# B&R Automation Studio project Parker_BMM_ST_V5_3147_V12 (part 4)

```iecst
(*Temperature fix and parameter type *)

TYPE
	Zones_Status_typ : 	STRUCT
		idxNotNormal : USINT;
		bNotNormal : BOOL;
		bAlarmHeatNormal : ARRAY[0..MAX_IDX_ZONE]OF BOOL;
		idxBroken : USINT;
		bBroken : BOOL; (*machine sensor broken*)
		SensorBroken : ARRAY[0..MAX_IDX_ZONE]OF BOOL; (*zone sensor broken*)
		bLowInternal : BOOL;
		idxLow : USINT;
		bLow : BOOL; (*machine alarm low*)
		AlmLow : ARRAY[0..MAX_IDX_ZONE]OF BOOL; (*zone alarm low*)
		idxHigh : USINT;
		bHigh : BOOL; (*machine alarm high*)
		AlmHigh : ARRAY[0..MAX_IDX_ZONE]OF BOOL; (*zone alarm high*)
		idxSwitchoff : USINT;
		bSwitchOff : BOOL; (*machine temperature high -switch off*)
		TempSwitchOff : ARRAY[0..MAX_IDX_ZONE]OF BOOL; (*temperature too high -- switch off*)
		idxFreeze : USINT;
		bFreeze : BOOL; (*machine heating exception*)
		TempFreeze : ARRAY[0..MAX_IDX_ZONE]OF BOOL; (*heating exception -- temperature freeze*)
		Tuning : ARRAY[0..MAX_IDX_ZONE]OF BOOL; (*zone is tuning*)
		TuneOk : ARRAY[0..MAX_IDX_ZONE]OF BOOL; (*zone tuning ok*)
		TuneStatus : ARRAY[0..MAX_IDX_ZONE]OF UINT; (*zone tune step and error feedback*)
		PreHeatingOk : ARRAY[0..MAX_IDX_ZONE]OF BOOL; (*zone pre-heating ok or not*)
		okToHeat : ARRAY[0..MAX_IDX_ZONE]OF BOOL; (*function need*)
		okToFree : ARRAY[0..MAX_IDX_ZONE]OF BOOL; (*function need*)
		okToFreeEnd : ARRAY[0..MAX_IDX_ZONE]OF BOOL; (*function need*)
		okToCool : ARRAY[0..MAX_IDX_ZONE]OF BOOL; (*function need*)
		okToCoolEnd : ARRAY[0..MAX_IDX_ZONE]OF BOOL; (*function need*)
		Out : ARRAY[0..MAX_IDX_ZONE]OF INT;
	END_STRUCT;
END_TYPE
```

### Global.var - Global variable
```iecst
(*global variables*)
VAR
	gAccuLinear : DCDT_typ;
	gAlarm : Alarm_typ;
	gAxisCtrl : ARRAY[0..MAX_AXIS_NUM] OF Axis_Ctrl_typ;
	gControlInfo : Control_Info_typ;
	gDS1119_Axis : ARRAY[0..MAX_AXIS_NUM] OF DS;
END_VAR
VAR RETAIN
	gExtruderA : Extruder_Ctrl_typ;
	gExtruderB : Extruder_Ctrl_typ;
	gExtruderC : Extruder_Ctrl_typ;
	gExtruderD : Extruder_Ctrl_typ := (0);
	gExtruderVisu : Extruder_Ctrl_typ;
	gH_IO : H_Zone_typ := (0);
END_VAR
VAR
	gHardWare : HardWare_typ;
END_VAR
VAR RETAIN
	gHeatingPlan : Heating_Plan_typ := (0);
END_VAR
VAR
	gImply : Imply_typ;
	gMachineFix : Machine_Fix_typ;
	gMachineIn : Machine_In_typ;
	gMachineInfo : Machine_Info_typ;
	gMachineOut : Machine_Out_typ;
	gMachinePara : Machine_Para_typ;
END_VAR
VAR RETAIN
	gMachineWorkDays : UDINT;
	gMachineStopDays : UDINT;
	gMachineWorkTime : UDINT;
	gMacOption : Machine_Option_typ;
	gBatchInfo : Batch_Info_typ;
END_VAR
VAR
	gMacTimer : Machine_Timer_typ;
	gPanelObj : Panel_Basic_typ;
	gPROCESS_info : Process_Status_typ;
	gPwd : Pwd_typ;
	gRecipeOperate : Recipe_Operate_typ;
	gScreenShot : ScreenShotObj_typ;
	gServoLinear : DCDT_typ;
END_VAR
VAR RETAIN
	gSPC_Current : SPC_Unit_typ;
	gT_Par : Temp_Ctrl_typ := (0);
END_VAR
VAR
	gThickData : Thick_Data_typ;
	gTempData : ARRAY[0..100] OF DINT;
	gThickFix : Thick_Fix_typ;
	gThickIO : Thick_IO_typ;
END_VAR
VAR RETAIN
	gThickProf : Profile_typ;
END_VAR
VAR
	gTKauto : task_status_type;
	gTKcalib : task_status_type;
	gTKmanual : task_status_type;
	gUSB_1 : USB_Device_typ;
	gUSB_2 : USB_Device_typ;
	gUserFix : User_Fix_typ;
	gUserFix_new : User_Fix_new_typ;
	gUserPara : User_Para_typ;
END_VAR
VAR RETAIN
	gCycleTimes : UDINT;
	gCycleTimesL : UDINT;
	gCycleTimesR : UDINT;
END_VAR
VAR CONSTANT
	LED_OFF : USINT := 0;
	LED_ON : USINT := 1;
	LED_QUICK_BLINK : USINT := 3;
	LED_SLOW_BLINK : USINT := 2;
END_VAR
VAR
	LMold : Mold_typ;
	RMold : Mold_typ;
END_VAR
(*Test Pump*)
VAR
	btnTesetPQ1 : BOOL;
	btnTesetPQ : BOOL;
END_VAR
(*Servo Axis*)
VAR
	gAxisClampL : ACP10AXIS_typ;
	gAxisClampR : ACP10AXIS_typ;
	gAxisCarriageL : ACP10AXIS_typ;
	gAxisCarriageR : ACP10AXIS_typ;
	gAxisBlowPinL : ACP10AXIS_typ;
	gAxisBlowPinR : ACP10AXIS_typ;
	gAxisBlowPin2L : ACP10AXIS_typ;
	gAxisBlowPin2R : ACP10AXIS_typ;
	gAxisTransferL : ACP10AXIS_typ;
	gAxisTransferR : ACP10AXIS_typ;
	gAxisUpDnL : ACP10AXIS_typ;
	gAxisUpDnR : ACP10AXIS_typ;
	gAxisExtrlift : ACP10AXIS_typ;
	gAxisThick : ACP10AXIS_typ;
END_VAR
(*Extruder Inverter Powerlink*)
VAR
	ExtruderA_Retain : {REDUND_UNREPLICABLE} Extruder_Basic_typ := (0); (*wzq*)
	ExtruderB_Retain : {REDUND_UNREPLICABLE} Extruder_Basic_typ := (0); (*wzq*)
	ExtruderC_Retain : Extruder_Basic_typ;
	ExtruderV_Retain : Extruder_Basic_typ;
	gExtruderACtrl : Inverter_Ctrl_typ;
	gExtruderBCtrl : Inverter_Ctrl_typ;
	gExtruderCCtrl : Inverter_Ctrl_typ;
	gExtruderVCtrl : Inverter_Ctrl_typ;
END_VAR
(*Robot Time*)
VAR
	LRobotCarriageTime : TOF_10ms;
	RobotCarriageTime : TOF_10ms;
	LRobotClampTime : TOF_10ms;
	RobotClampTime : TOF_10ms;
END_VAR
(*Insert your comment here.*)
VAR
	LRobotClampTimePara : UDINT;
	RobotClampTimePara : UDINT;
	LRobotCarriageTimePara : UDINT;
	RobotCarriageTimePara : UDINT;
	usScaleIndex : USINT;
	gLClampOpnFlag_Calib : USINT;
	gRClampOpnFlag_Calib : USINT;
	ParisonSacleDown : DINT;
	ParisonSacleUp : DINT;
	ParisonSacleDown_Old : DINT;
	ParisonSacleUp_Old : DINT;
	ParisonSacleDownFlag : BOOL;
	ParisonSacleUpFlag : BOOL;
	ParisonSacleDownFlag_Old : BOOL;
	ParisonSacleUpFlag_Old : BOOL;
	gLevelTooLow : BOOL;
	gExtruderTempLow_HMIFlag : BOOL;
	gTempfirstHeatOK : DINT;
	gTempfirstHeatOK_Flag : BOOL;
	gPasswordLogout : BOOL;
	gAcs380Ctrl : Acs380Ctl_type;
	gEnableAll_HMI : BOOL;
	gDisableAll_HMI : BOOL;
	gExtruderHMI_Enable : ARRAY[0..NUM_ACS380_MINUS_ONE] OF BOOL;
END_VAR
VAR CONSTANT
	NUM_ACS380_MINUS_ONE : USINT := 4; (*Acs380数量-1*)
END_VAR
VAR
	ExIndex : USINT;
	gExSPC : ARRAY[0..19] OF ExSPC_typ;
	gExSPC_Clear : BOOL;
	gAxisPwr : ACP10AXIS_typ;
	gMotorTrace : MotorTrace_typ;
	gAxisCarriageR_1 : ACP10AXIS_typ;
END_VAR
```

### Library Logical/Libraries/SimpFun (IEC, version 2.10.0) - Get time function library
Depends on: AsIO, AsString, AsTime, runtime

#### DateTimeString.st
```iecst
FUNCTION_BLOCK DateTimeString
(* Implementation of ST_DateTimeString *)

(*
//******************************************************************************************************//
//		 B & R - Bernecker and Rainer China 		              										              //
//******************************************************************************************************//
// Library Name:	SimpFun																			                       //
// Function Name:	DateTimeString																		                    //
// Autor:			B&R 						      	  										                          //
//------------------------------------------------------------------------------------------------------//
// Description: 	Print Different type Date and Time									  				              //
//-------------------------------------------------------------------------------------------------------//

//-------------------------------------------------------------------------------------------------------//
//	History:	6.Nov.2008	 V1.00														                                 //
//				V1.00: Just 24 hour time mode															                     //
//*******************************************************************************************************//

//*******************************************************************************************************//
//	<|> Variable to control this task:																	                  //
//		Name							Typ					Description									                     //
//		strYYYY							STRING[4]			Save Year as STRING	type			                     //
//		strMonthM						STRING[2]			Save Month as STRING type			                     //
//		strDD							STRING[2]			Save Day as STRING type						                  //
//		strHH							STRING[2]			Save Hour as STRING type					                  //
//		strMinuteM						STRING[2]			Save Minute as STRING type				                  //
//		strSS							STRING[2]			Save Second as STRING type					                  //
//		flagAMPM						BOOL				current time is AM or PM:0=AM,1=PM			                  //
//*******************************************************************************************************//

//*******************************************************************************************************//
//  Others:																								                        //
//		V1.00:																							                        //
//			Date_Mode																					                        //
//				1:		USA date format -- DateMM-DD-YYYY_TimeHH-MM-SS								                  //
//				2:		Asia DATE format -- DateYYYY-MM-DD_TimeHH-MM-SS								                  //
//				others:	Default format -- DateDD-MM-YYYY_TimeHH-MM-SS							                  //
//*******************************************************************************************************//
*)

IF (enable = 1) THEN

	DTGetTime_0.enable := 1;
	DTGetTime_0();

	DT_TO_DTStructure(DTGetTime_0.DT1, ADR(currentTime));

	strcpy(ADR(DisplayString),ADR('Date'));								(* DisplayString = "Date" *)

	itoa(currentTime.year, ADR(strYYYY));								(* string -- "YYYY" *)
	itoa(currentTime.month, ADR(strMonthM));							(* string -- "MM: month" *)
	itoa(currentTime.day, ADR(strDD));									(* string -- "DD" *)

	CASE Date_Mode OF
		1:		(* USA date format -- MM-DD-YYYY *)

			(***** ADD MM   Month *****)
			IF currentTime.month <= 9 THEN
				strcat(ADR(DisplayString), ADR('0'));					(* DisplayString = "Date0" *)
			END_IF
			strcat(ADR(DisplayString), ADR(strMonthM));					(* DisplayString = "DateMM" *)
			strcat(ADR(DisplayString), ADR('-'));						(* DisplayString = "DateMM-" *)

			(***** ADD DD *****)
			IF currentTime.day <= 9 THEN
				strcat(ADR(DisplayString), ADR('0'));					(* DisplayString = "DateMM-0" *)
			END_IF
			strcat(ADR(DisplayString), ADR(strDD));						(* DisplayString = "DateMM-DD" *)
			strcat(ADR(DisplayString), ADR('-'));						(* DisplayString = "DateMM-DD-" *)

			(***** ADD YYYY *****)
			strcat(ADR(DisplayString), ADR(strYYYY));					(* DisplayString = "DateMM-DD-YYYY" *)

		2:		(* Asia date format -- YYYY-MM-DD *)

			(***** ADD YYYY *****)
			strcat(ADR(DisplayString), ADR(strYYYY));					(* DisplayString = "DateYYYY" *)
			strcat(ADR(DisplayString), ADR('-'));						(* DisplayString = "DateYYYY-" *)

			(***** ADD MM   Month *****)
			IF currentTime.month <= 9 THEN
				strcat(ADR(DisplayString), ADR('0'));					(* DisplayString = "DateYYYY-0" *)
			END_IF
			strcat(ADR(DisplayString), ADR(strMonthM));					(* DisplayString = "DateYYYY-MM" *)
			strcat(ADR(DisplayString), ADR('-'));						(* DisplayString = "DateYYYY-MM-" *)

			(***** ADD DD *****)
			IF currentTime.day <= 9 THEN
				strcat(ADR(DisplayString), ADR('0'));					(* DisplayString = "DateYYYY-MM-0" *)
			END_IF
			strcat(ADR(DisplayString), ADR(strDD));						(* DisplayString = "DateYYYY-MM-DD" *)

		ELSE	(* Default format -- DD-MM-YYYY *)

			(***** ADD DD *****)
			IF currentTime.day <= 9 THEN
				strcat(ADR(DisplayString), ADR('0'));					(* DisplayString = "Date0" *)
			END_IF
			strcat(ADR(DisplayString), ADR(strDD));						(* DisplayString = "DateDD" *)
			strcat(ADR(DisplayString), ADR('-'));						(* DisplayString = "DateDD-" *)

			(***** ADD MM   Month *****)
			IF currentTime.month <= 9 THEN
				strcat(ADR(DisplayString), ADR('0'));					(* DisplayString = "DateDD-0" *)
			END_IF
			strcat(ADR(DisplayString), ADR(strMonthM));					(* DisplayString = "DateDD-MM" *)
			strcat(ADR(DisplayString), ADR('-'));						(* DisplayString = "DateDD-MM-" *)

			(***** ADD YYYY *****)
			strcat(ADR(DisplayString), ADR(strYYYY));					(* DisplayString = "DateDD-MM-YYYY" *)

	END_CASE

	strcat(ADR(DisplayString),ADR('_Time'));							(* DisplayString = "DateDD-MM-YYYY_Time" *)

	itoa(currentTime.minute, ADR(strMinuteM));							(* string -- "MM: minute" *)
	itoa(currentTime.second, ADR(strSS));								(* string -- "SS" *)

	(***** ADD HH : 24 Hour mode*****)
		IF currentTime.hour <= 9 THEN
			strcat(ADR(DisplayString), ADR('0'));						(* DisplayString = "DateDD-MM-YYYY_Time0" *)
		END_IF
		itoa(currentTime.hour, ADR(strHH));								(* string -- "HH" *)
		strcat(ADR(DisplayString), ADR(strHH));							(* DisplayString = "DateDD-MM-YYYY_TimeHH" *)
	END_IF
	strcat(ADR(DisplayString), ADR('-'));								(* DisplayString = "DateDD-MM-YYYY_TimeHH-" *)

	(***** ADD MM   minute *****)
	IF currentTime.minute <= 9 THEN
		strcat(ADR(DisplayString), ADR('0'));							(* DisplayString = "DateDD-MM-YYYY_TimeHH-0" *)
	END_IF
	strcat(ADR(DisplayString), ADR(strMinuteM));						(* DisplayString = "DateDD-MM-YYYY_TimeHH-MM" *)
	strcat(ADR(DisplayString), ADR('-'));								(* DisplayString = "DateDD-MM-YYYY_TimeHH-MM-" *)

	(***** ADD SS *****)
	IF currentTime.second <= 9 THEN
		strcat(ADR(DisplayString), ADR('0'));							(* DisplayString = "DateDD-MM-YYYY_TimeHH-MM-0" *)
	END_IF
	strcat(ADR(DisplayString), ADR(strSS));								(* DisplayString = "DateDD-MM-YYYY_TimeHH-MM-SS" *)

	StringLength := strlen(ADR(DisplayString));							(* Output StringLength -- length of the DisplayString *)

END_FUNCTION_BLOCK
```

#### IOForcingOperate.st
```iecst
FUNCTION_BLOCK IOForcingOperate
(* Implementation of IOForcingOperate *)

(*
//******************************************************************************************************//
//		 B & R - Bernecker and Rainer China 		              										              //
//******************************************************************************************************//
// Library Name:	SimpFun																			                       //
// Function Name:	IOForcingOperate																	                    //
// Autor:			B&R 						      	  										                          //
//------------------------------------------------------------------------------------------------------//
// Description: 	operate IO: Enable/disable 		 									  				              //
//------------------------------------------------------------------------------------------------------//

//------------------------------------------------------------------------------------------------------//
//	History:	 	23.Nov.2008	 V1.00														                             //

//******************************************************************************************************//

//******************************************************************************************************//
//	<|> Variable to control this task:																	                 //
//		Name						Typ						Description									                    //
//		AsIOSetForceValue_0			| AsIOSetForceValue 	| Set force value							              //
//		AsIOEnableForcing_0			| AsIOEnableForcing 	| Enable force value						              //
//		AsIODisableForcing_0		| AsIODisableForcing 	| Disable forceing							           //

//******************************************************************************************************//

//******************************************************************************************************//
//  Others:																								                       //
//		V1.00:																							                       //
			be careful: make sure EnableForcing and DisableForcing, only one is true.
//		Name						Typ						Description									                    //
		IN:
//			enable					| BOOL					| enable this function						              //
//			EnableForcing			| BOOL					| =1:this function use to enable forcing	           //
//			Value					| UDINT					| the forcing value							                 //
//			DisableForcing			| BOOL					| =1:this function use to disable forcing	           //
		OUT:
//			status					| UINT					| =0: no error								                 //
//			InForcing				| USINT					| =0: No forcing							                 //
//															  =1: Forcing to zero						                    //
//															  =2: Forcing to one						                       //

//******************************************************************************************************//
*)

IF (enable = 1) THEN
	CASE (step) OF
		0:			(* init step *)
			status := 65535;
			IF (EnableForcing = 1) THEN								(* Enable Forcing *)
				step := 10;
			ELSIF (DisableForcing = 1) THEN
				step := 30;											(* Disable Forcing *)
			END_IF

		10:			(* set force value *)
			AsIOSetForceValue_0.enable     := 1;
			AsIOSetForceValue_0.pDatapoint := ADR(DataPoint);		(* Pointer to the I/O data point name *)
			AsIOSetForceValue_0.value      := Value;

			AsIOSetForceValue_0();

			IF (AsIOSetForceValue_0.status <> 65535) THEN
				IF (AsIOSetForceValue_0.status = 0) THEN
					step := 20;
				ELSE
					status := AsIOSetForceValue_0.status;
					step := 200;									(* Error *)
				END_IF
			END_IF

		20:			(* Enable forcing *)
			AsIOEnableForcing_0.enable := 1;
			AsIOEnableForcing_0.pDatapoint := ADR(DataPoint);

			AsIOEnableForcing_0();

			IF (AsIOEnableForcing_0.status <> 65535) THEN
				IF (AsIOEnableForcing_0.status = 0) THEN
					IF (Value = 0) THEN
						InForcing := 1;
					ELSE
						InForcing := 2;
					END_IF
					step := 100;									(* Enable forcing ok *)

				ELSE
					status := AsIOEnableForcing_0.status;
					step := 200;									(* Error *)

				END_IF
			END_IF

		30:			(* Disable forcing *)
			AsIODisableForcing_0.enable := 1;
			AsIODisableForcing_0.pDatapoint := ADR(DataPoint);

			AsIODisableForcing_0();

			IF (AsIODisableForcing_0.status <> 65535) THEN
				IF (AsIODisableForcing_0.status = 0) THEN
					InForcing := 0;
					step := 100;									(* Disable forcing ok *)
				ELSE
					status := AsIODisableForcing_0.status;
					step := 200;									(* Error *)
				END_IF
			END_IF

		100:		(* Operator OK *)
			status := 0;
			step := 0;

		200: 		(* Error step *)
			(* the error number has record in status *)
			step := 0;

	END_CASE
END_IF
END_FUNCTION_BLOCK
```

#### Scaler_ActZone.st
```iecst
FUNCTION_BLOCK Scaler_ActZone
(* Implementation of Scaler_ActZone *)

IF Enable = 1 THEN
	IF (MaxInV <= MinInV) OR (MaxOutV <= MinOutV) OR (ActZoneMaxV <= ActZoneMinV) THEN

		status := 1;							(* Parameter Error: MaxInV/MaxOutV/ActZoneMaxV must larger than MinInV/MinOutV/ActZoneMinV *)
	ELSIF (ActZoneMinV < MinInV) OR (MaxInV < ActZoneMaxV) THEN
		status := 2;							(* Parameter Error: [ActZoneMinV, ActZoneMaxV] must be loacaled in [MinInV, MaxInV] *)
	ELSIF (Mode_Current = 0) AND ((MinOutV < -10) OR (MaxOutV > 10)) THEN
		status := 3;							(* Parameter Error: For Voltage Output, MaxInV and MinInV must be localed in [-10, 10] *)
	ELSIF (Mode_Current = 1) AND ((MinOutV < -20) OR (MaxOutV > 20)) THEN
		status := 4;							(* Parameter Error: For Current Output, MaxInV and MinInV must be localed in [-20, 20] *)
	ELSE										(* Parameter Correct *)
		status := 0;

		IF (SV < ActZoneMinV) THEN
			IF (Mode_Current = 0) THEN
				Out := REAL_TO_INT(INT_TO_REAL(MinOutV)*32767/10);
			ELSE
				Out := REAL_TO_INT(INT_TO_REAL(MinOutV)*32767/20);
			END_IF
		ELSIF (SV > ActZoneMaxV) THEN
			IF (Mode_Current = 0) THEN
				Out := REAL_TO_INT(INT_TO_REAL(MinOutV)*32767/10);
			ELSE
				Out := REAL_TO_INT(INT_TO_REAL(MinOutV)*32767/20);
			END_IF
		ELSE
			IF (Mode_Current = 0) THEN
				Out := REAL_TO_INT(((INT_TO_REAL(MaxOutV) - MinOutV)*(SV - MinInV)/(MaxInV - MinInV) + MinOutV)*32767/10);
			ELSE
				Out := REAL_TO_INT(((INT_TO_REAL(MaxOutV) - MinOutV)*(SV - MinInV)/(MaxInV - MinInV) + MinOutV)*32767/20);
			END_IF
		END_IF
	END_IF
END_IF
END_FUNCTION_BLOCK
```

#### SimpFun.fun
```iecst
FUNCTION_BLOCK DateTimeString
VAR
		DTGetTime_0	:DTGetTime;
		currentTime	:DTStructure;
		strYYYY	:STRING[4];
		strDD	:STRING[2];
		strHH	:STRING[2];
		strSS	:STRING[2];
		strMonthM	:STRING[2];
		strMinuteM	:STRING[2];
	END_VAR
	VAR_INPUT
		enable	:BOOL;
		Date_Mode	:USINT;
	END_VAR
	VAR_OUTPUT
		DisplayString	:STRING[80];
		StringLength	:UINT;
	END_VAR
END_FUNCTION_BLOCK
FUNCTION_BLOCK IOForcingOperate
VAR
		step	:USINT;
		AsIOSetForceValue_0	:AsIOSetForceValue;
		AsIOEnableForcing_0	:AsIOEnableForcing;
		AsIODisableForcing_0	:AsIODisableForcing;
	END_VAR
	VAR_INPUT
		enable	:BOOL;
		DataPoint	:STRING[80];
		EnableForcing	:BOOL;
		Value	:UDINT;
		DisableForcing	:BOOL;
	END_VAR
	VAR_OUTPUT
		status	:UINT;
		InForcing	:USINT;
	END_VAR
END_FUNCTION_BLOCK
FUNCTION_BLOCK Scaler_ActZone
VAR_INPUT
		Enable	:BOOL;
		MaxInV	:INT;
		MinInV	:INT;
		ActZoneMaxV	:INT;
		ActZoneMinV	:INT;
		MaxOutV	:INT;
		MinOutV	:INT;
		SV	:INT;
		Mode_Current	:BOOL;
	END_VAR
	VAR_OUTPUT
		Out	:INT;
		status	:UINT;
	END_VAR
END_FUNCTION_BLOCK
```

### Program Logical/In_Out/tk1_in (ANSIC) - task 1 fast input

#### tk1_in.c
```c
/********************************************************************
 * COPYRIGHT --  B&R China
 ********************************************************************
 * Program: tk1_in
 * File: tk1_in.c
 * Author: lijianjun
 * Created: March 06, 2013
 ********************************************************************
 * Implementation of program tk1_in --- task 1# input
 ********************************************************************/

#include <bur/plctypes.h>
#include <string.h>

#ifdef _DEFAULT_INCLUDES
#include <AsDefault.h>
#endif

#include "edge.h"               /*edge function                         */

/*************************************************************************************
     	        		I N I T U P  O F   T H E   T A S K
*************************************************************************************/
_INIT void init ( void )
{
	RTInfo_Task.enable = 1;
	RTInfo(&RTInfo_Task);

	tTask = RTInfo_Task.cycle_time/1000.0/1000.0;		/*  from us ---> s  */

	memset(&LCarriageFilter,0,sizeof(LCarriageFilter));
	LCarriageFilter.enable = 1;
	LCarriageFilter.Times  = 20;

	memset(&RCarriageFilter,0,sizeof(RCarriageFilter));
	RCarriageFilter.enable = 1;
	RCarriageFilter.Times  = 20;

	memset(&LClampFilter,0,sizeof(LClampFilter));
	LClampFilter.enable = 1;
	LClampFilter.Times  = 20;

	memset(&RClampFilter,0,sizeof(RClampFilter));
	RClampFilter.enable = 1;
	RClampFilter.Times  = 20;

	memset(&LBlowpinFilter,0,sizeof(LBlowpinFilter));
	LBlowpinFilter.enable = 1;
	LBlowpinFilter.Times  = 20;

	memset(&RBlowpinFilter,0,sizeof(RBlowpinFilter));
	RBlowpinFilter.enable = 1;
	RBlowpinFilter.Times  = 20;

	memset(&ServoFilter,0,sizeof(ServoFilter));
	ServoFilter.enable = 1;
	ServoFilter.Times  = 10;

	lPT2_MeltP_A.Ts = tTask;
	lPT2_MeltP_A.T1 = tTask * 10;
	lPT2_MeltP_A.T2 = tTask * 10;

	lPT2_MeltP_B.Ts = tTask;
	lPT2_MeltP_B.T1 = tTask * 10;
	lPT2_MeltP_B.T2 = tTask * 10;

	/*2018.7.10 Albert*/
	/*ACC Pressure*/
	IPT2_ACC_P.Ts = tTask;
	IPT2_ACC_P.T1 = tTask * 10;
	IPT2_ACC_P.T2 = tTask * 10;

	/* differentiator for evaluating the actual speed */
	vActHydDT2ExtrA.Ts = tTask;	/* cycle time 0.002s 			  */
	vActHydDT2ExtrA.Tv = 60.0; 	/* derivative time constant [s]   */
	vActHydDT2ExtrA.T1 = 2.0; 	   /* filter time constant 1 : 0.1s */
	vActHydDT2ExtrA.T2 = 2.0; 	   /* filter time constant 2 : 0.1s */

	/* differentiator for evaluating the actual speed */
	vActHydDT2ExtrB.Ts = tTask;	/* cycle time 0.002s 			  */
	vActHydDT2ExtrB.Tv = 60.0; 	/* derivative time constant [s]   */
	vActHydDT2ExtrB.T1 = 2.0; 	   /* filter time constant 1 : 0.1s */
	vActHydDT2ExtrB.T2 = 2.0; 	   /* filter time constant 2 : 0.1s */

	/* differentiator for evaluating the actual speed */
	vActHydDT2ExtrC.Ts = tTask;	/* cycle time 0.002s 			  */
	vActHydDT2ExtrC.Tv = 60.0; 	/* derivative time constant [s]   */
	vActHydDT2ExtrC.T1 = 2.0; 	   /* filter time constant 1 : 0.1s */
	vActHydDT2ExtrC.T2 = 2.0; 	   /* filter time constant 2 : 0.1s */

	/* differentiator for evaluating the actual speed */
	vActHydDT2ExtrVisu.Ts = tTask;	/* cycle time 0.002s 			  */
	vActHydDT2ExtrVisu.Tv = 60.0; 	/* derivative time constant [s]   */
	vActHydDT2ExtrVisu.T1 = 2.0; 	   /* filter time constant 1 : 0.1s */
	vActHydDT2ExtrVisu.T2 = 2.0; 	   /* filter time constant 2 : 0.1s */

	/*Servo Flux linear*/
	LinSplineOilFlux.enable = 1;
	LinSplineOilFlux.NbNodes = 2;
	LinSplineOilFlux.Smooth = 0;
	LinSplineOilFlux.Rness = 100.0;
	LinSplineOilFlux.Invert = 0;
	LinSplineOilFlux.DisMode = 0;
	LinSplineOilFlux.pNodeVec = &OilFluxNode[0];
	LinSplineOilFlux.Update	=	1;

}/* _INIT void init ( void )  */
/**************************************************************************************
****				C Y C L I C   P A R T   O F   T H E   T A S K  				           ****
**************************************************************************************/
_CYCLIC void cyclic ( void )
{
	/* ------------- thickness LVDT ------------- */
		if(gHardWare.AI4632_2[0]  >= 0)
		{
			ServoFilter.u= gHardWare.AI4632_2[0];
			HydMovAvgFlt(&ServoFilter);
		}
		gServoLinear.Current = ServoFilter.y;

	/* -------------  right carriage LVDT ------------- */
	//		if(gHardWare.AI4632_1[3] >= 0)
	//		{
	//			RCarriageFilter.u = gHardWare.AI4632_1[3];
	//			HydMovAvgFlt(&RCarriageFilter);
	//		}
	//
	//		RMold.Carriage.As = RCarriageFilter.y;

	/* -------------  left carriage LVDT ------------- */
	//		if(gHardWare.AI4632_1[2] >= 0)
	//		{
	//			LCarriageFilter.u = gHardWare.AI4632_1[2];
	//			HydMovAvgFlt(&LCarriageFilter);
	//		}
	//
	//		LMold.Carriage.As = LCarriageFilter.y;

	/* -------------  right clamp LVDT  ------------- */
	if(gHardWare.AI4632_1[0]>= 0)
	{
		RClampFilter.u = gHardWare.AI4632_1[0];
		HydMovAvgFlt(&RClampFilter);
	}

	if(ACTUATOR_HYD == gMachineFix.MoldR.Clamp.eActuatorType)
	{
		RMold.Clamp.As  = RClampFilter.y;
	}

	/* -------------  left clamp LVDT  ------------- */
	if(gHardWare.AI4632_1[1] >= 0)
	{
		LClampFilter.u = gHardWare.AI4632_1[1];
		HydMovAvgFlt(&LClampFilter);
	}
	if(ACTUATOR_HYD == gMachineFix.MoldR.Clamp.eActuatorType)
	{
		LMold.Clamp.As  = LClampFilter.y;
	}

	/* -------------  right blowpin LVDT  ------------- */
	if(gHardWare.AI4632_2[1]>= 0)
	{
		RBlowpinFilter.u = gHardWare.AI4632_2[1];
		HydMovAvgFlt(&RBlowpinFilter);
	}

	if(ACTUATOR_HYD == gMachineFix.MoldR.BlowPin.eActuatorType)
	{
		RMold.BlowPin.As  = RBlowpinFilter.y;
	}

//	/* -------------  left blowpin LVDT  ------------- */
//	if(gHardWare.AI4632_1[1] >= 0)
//	{
//		LBlowpinFilter.u = gHardWare.AI4632_1[1];
//		HydMovAvgFlt(&LBlowpinFilter);
//	}
//	if(ACTUATOR_HYD == gMachineFix.MoldR.BlowPin.eActuatorType)
//	{
//		LMold.BlowPin.As  = LBlowpinFilter.y;
//	}

	/* ----------------- A extruder speed ----------------- */
	/*------------------*/
	/*-----DI Pulse-----*/

	//	gExtruderA.diActRPM = gHardWare.DI9371_3[6];
	//	if(1 == EDGEPOS(gExtruderA.diActRPM,DISpeedExtrA))
	//	{
	//		RotatespeedExtrA = RotatespeedExtrA + 1;
	//	}
	//
	//	DISpeedExtrA = gExtruderA.diActRPM;
	//
	//	vActHydDT2ExtrA.u = RotatespeedExtrA * 0.1;
	//
	//	if(vActHydDT2ExtrA.u < 0)vActHydDT2ExtrA.u = -vActHydDT2ExtrA.u;
	//
	//	/* call function block */
	//	HydDT2(&vActHydDT2ExtrA);
	//
	//	gExtruderA.ActRPM = vActHydDT2ExtrA.y;
	//	if(gExtruderA.ActRPM < 0)gExtruderA.ActRPM= -gExtruderA.ActRPM;

	//	gExtruderA.aiCurrent = gHardWare.AI4632_1[2];
	//	gExtruderA.aiMeltPressure = gHardWare.AI4632_4[0];

	/*-------------------------*/
	/*------AI  0 ~ 32767------*/
	gExtruderA.aiActRPM = gHardWare.AI4632_2[0];

	/* ----------------- B extruder speed ----------------- */

	/*------------------*/
	/*-----DI Pulse-----*/
	//	gExtruderB.diActRPM = gHardWare.DI9371_3[0];
	//	if(1 == EDGEPOS(gExtruderB.diActRPM,DISpeedExtrB))
	//	{
	//		RotatespeedExtrB = RotatespeedExtrB + 1;
	//	}
	//
	//	DISpeedExtrB = gExtruderB.diActRPM;
	//
	//	vActHydDT2ExtrB.u = RotatespeedExtrB * 0.1;
	//
	//	if(vActHydDT2ExtrB.u < 0)vActHydDT2ExtrB.u = -vActHydDT2ExtrB.u;
	//
	//	/* call function block */
	//	HydDT2(&vActHydDT2ExtrB);
	//
	//	gExtruderB.ActRPM = vActHydDT2ExtrB.y;
	//	if(gExtruderB.ActRPM < 0)gExtruderB.ActRPM = -gExtruderB.ActRPM;

	//	gExtruderB.aiActRPM  = gHardWare.AI4632_4[3];
	//	gExtruderB.aiCurrent = gHardWare.AI4632_1[3];

	/*-------------------------*/
	/*------AI  0 ~ 32767------*/
	gExtruderB.aiActRPM = gHardWare.AI4632_3[2];

	/* ----------------- C extruder speed ----------------- */

	/*------------------*/
	/*-----DI Pulse-----*/
	//	if(1 == EDGEPOS(gExtruderC.diActRPM,DISpeedExtrC))
	//	{
	//		RotatespeedExtrC = RotatespeedExtrC + 1;
	//	}
	//
	//	DISpeedExtrC = gExtruderC.diActRPM;
	//
	//	vActHydDT2ExtrC.u = RotatespeedExtrC * 0.1;
	//
	//	if(vActHydDT2ExtrC.u < 0)vActHydDT2ExtrC.u = -vActHydDT2ExtrC.u;
	//
	//	/* call function block */
	//	HydDT2(&vActHydDT2ExtrC);
	//
	//	gExtruderC.ActRPM = vActHydDT2ExtrC.y;
	//	if(gExtruderC.ActRPM < 0)gExtruderC.ActRPM = -gExtruderC.ActRPM;

	/*-------------------------*/
	/*------AI  0 ~ 32767------*/
	gExtruderC.aiActRPM = gHardWare.AI4632_3[3];

	/* ----------------- D extruder speed ----------------- */

	/*------------------*/
	/*-----DI Pulse-----*/
	//	gExtruderD.diActRPM = gHardWare.DI9371_3[7];
	//	if(1 == EDGEPOS(gExtruderD.diActRPM,DISpeedExtrD))
	//	{
	//		RotatespeedExtrD = RotatespeedExtrD + 1;
	//	}
	//
	//	DISpeedExtrD = gExtruderD.diActRPM;
	//
	//	vActHydDT2ExtrD.u = RotatespeedExtrD * 0.1;
	//
	//	if(vActHydDT2ExtrD.u < 0)vActHydDT2ExtrD.u = -vActHydDT2ExtrD.u;
	//
	//	/* call function block */
	//	HydDT2(&vActHydDT2ExtrD);
	//
	//	gExtruderD.ActRPM = vActHydDT2ExtrD.y;
	//	if(gExtruderD.ActRPM < 0)gExtruderD.ActRPM = -gExtruderD.ActRPM;
	//
	//	gExtruderD.aiActRPM  = gHardWare.AI4632_4[0];
	//	gExtruderD.aiCurrent = gHardWare.AI4632_4[0];

	/*-------------------------*/
	/*------AI  0 ~ 32767------*/
	gExtruderD.aiActRPM = gHardWare.AI4632_3[0];

	/* ----------------- Visual extruder speed ----------------- */

	/*------------------*/
	/*-----DI Pulse-----*/
	//	gExtruderVisu.diActRPM = gHardWare.DI9371_3[7];
	//	if(1 == EDGEPOS(gExtruderVisu.diActRPM,DISpeedExtrVisu))
	//	{
	//		RotatespeedExtrVisu = RotatespeedExtrVisu + 1;
	//	}
	//
	//	DISpeedExtrVisu = gExtruderVisu.diActRPM;
	//
	//	vActHydDT2ExtrVisu.u = RotatespeedExtrVisu * 0.1;
	//
	//	if(vActHydDT2ExtrVisu.u < 0)vActHydDT2ExtrVisu.u = -vActHydDT2ExtrVisu.u;
	//
	//	/* call function block */
	//	HydDT2(&vActHydDT2ExtrVisu);
	//
	//	gExtruderVisu.ActRPM = vActHydDT2ExtrVisu.y;
	//	if(gExtruderVisu.ActRPM < 0)gExtruderVisu.ActRPM = -gExtruderD.ActRPM;
	//
	//	gExtruderVisu.aiActRPM  = gHardWare.AI4632_4[0];
	//	gExtruderVisu.aiCurrent = gHardWare.AI4632_4[0];

	/*-------------------------*/
	/*------AI  0 ~ 32767------*/
	gExtruderVisu.aiActRPM = gHardWare.AI4632_3[1];

	/* ------------- A extruder melt pressure ------------- */
	if(0 == gMachineFix.ExtruderA.MeltP10V)gMachineFix.ExtruderA.MeltP10V = 8.0;

	lPT2_MeltP_A.u = gExtruderA.aiMeltPressure;

	/* call function block */
	HydPT2(&lPT2_MeltP_A);

	if((gMachineFix.ExtruderA.MeltP10V - gMachineFix.ExtruderA.MeltP0V) != 0.0)
	{
		gExtruderA.MeltPressure = (lPT2_MeltP_A.y/3276.7 - gMachineFix.ExtruderA.MeltP0V)* 560.0 /(gMachineFix.ExtruderA.MeltP10V - gMachineFix.ExtruderA.MeltP0V);
	}

	/* ------------- B extruder melt pressure ------------- */
	if(0 == gMachineFix.ExtruderB.MeltP10V)gMachineFix.ExtruderB.MeltP10V = 8.0;

	lPT2_MeltP_B.u = gExtruderB.aiMeltPressure;

	/* call function block */
	HydPT2(&lPT2_MeltP_B);

	if((gMachineFix.ExtruderB.MeltP10V - gMachineFix.ExtruderB.MeltP0V) != 0.0)
	{
		gExtruderB.MeltPressure = (lPT2_MeltP_B.y/3276.7 - gMachineFix.ExtruderB.MeltP0V)* 560.0 /(gMachineFix.ExtruderB.MeltP10V - gMachineFix.ExtruderB.MeltP0V);
	}
	/* ----------------------------------------- */
	/* ------------- ACC pressure ------------- */
	/* ----------------------------------------- */

	IPT2_ACC_P.u = gHardWare.AI4632_1[2];

	/* call function block */
	HydPT2(&IPT2_ACC_P);

	//	gMachineInfo.OilAccuPressure = (IPT2_ACC_P.y/32767) * gMachineFix.OilAccu.AccuPressure10V;
	/*--------------------------------------------------------------------------------------------------------------------*/
	//	if ((1==gMachineIn.OilPumpOk_DI && 1==gMachineInfo.OilPumpDelayDone && 0== gMachineInfo.Auto)) //ipis0222 Pump start finish
	//	{
	//		if(IPT2_ACC_P.y !=0)
	//		{
	//			if(1==	gMachineInfo.bAccuPumpCalib)
	//			{
	//				gUserPara.AccuPressure_Calib = gMachineFix.OilAccu.AccuPressure10V/IPT2_ACC_P.y;
	//			}
	//		}
	//	}
	//	gMachineInfo.OilAccuPressure = IPT2_ACC_P.y*gUserPara.AccuPressure_Calib;
	/*--------------------------------------------------------------------------------------------------------------------*/
	if (1 == gMacOption.OilPumpStartMode)
	{
		if ((1==gMachineIn.OilPumpOk_DI && 1==gMachineInfo.OilPumpDelayDone && 0== gMachineInfo.Auto)) //ipis0222 Pump start finish
		{
			if(IPT2_ACC_P.y !=0)
			{
				if(1==	gMachineInfo.bAccuPumpCalib)
				{
					//	gUserPara.AccuPressure_Calib = gMachineFix.OilAccu.AccuPressure10V/IPT2_ACC_P.y;
					//gUserPara.AccuPressure_Calib = IPT2_ACC_P.y;
					gUserFix_new.AccuPressure_Calib = IPT2_ACC_P.y;
				}
			}
		}
	}
	else
	{
		if ((1==gMachineIn.OilPumpOk_DI && 0== gMachineInfo.Auto)) //ipis0222 Pump start finish
		{
			if(IPT2_ACC_P.y !=0)
			{
				if(1==	gMachineInfo.bAccuPumpCalib)
				{
					//	gUserPara.AccuPressure_Calib = gMachineFix.OilAccu.AccuPressure10V/IPT2_ACC_P.y;
					//gUserPara.AccuPressure_Calib = IPT2_ACC_P.y;
					gUserFix_new.AccuPressure_Calib = IPT2_ACC_P.y;

				}
			}
		}
	}
	//	if ((1==gMachineIn.OilPumpOk_DI && 1==gMachineInfo.OilPumpDelayDone && 0== gMachineInfo.Auto)) //ipis0222 Pump start finish
	//	{
	//		if(IPT2_ACC_P.y !=0)
	//		{
	//			if(1==	gMachineInfo.bAccuPumpCalib)
	//			{
	//				//	gUserPara.AccuPressure_Calib = gMachineFix.OilAccu.AccuPressure10V/IPT2_ACC_P.y;
	//				//gUserPara.AccuPressure_Calib = IPT2_ACC_P.y;
	//				gUserFix_new.AccuPressure_Calib = IPT2_ACC_P.y;
	//
	//			}
	//		}
	//
	//
	//	}
	if ((0== gMachineInfo.Auto)) //ipis0222 Pump start finish
	{
		if(1==	gMachineInfo.bAccuPumpMinCalib)
		{
			//	gUserPara.AccuPumpMinCalib = IPT2_ACC_P.y;
			gUserFix_new.AccuPumpMinCalib = IPT2_ACC_P.y;
		}
	}
	if (IPT2_ACC_P.y-gUserFix_new.AccuPumpMinCalib >=0)
	{
		if (0!=(gUserFix_new.AccuPressure_Calib-gUserFix_new.AccuPumpMinCalib))  //ipis1207
		{
			gMachineInfo.OilAccuPressure=(IPT2_ACC_P.y-gUserFix_new.AccuPumpMinCalib)*((gMachineFix.OilAccu.AccuPressure10V-gUserFix_new.AccuPressure0V)/(gUserFix_new.AccuPressure_Calib-gUserFix_new.AccuPumpMinCalib));
		}
	}
	else
	{
		gMachineInfo.OilAccuPressure =0;
	}

	/*--------------------------------------------------------------------------------------------------------------------*/

	/* ------------------------------------------------------ */
	/* ------------- Extrlift ACC pressure ------------------ */
	/* ------------------------------------------------------ */

	IPT2_ACC_Extrlift_P.u = gHardWare.AI4632_1[1];

	/* call function block */
	HydPT2(&IPT2_ACC_Extrlift_P);

	if (1 == gMacOption.OilPumpStartMode)
	{
		if ((1==gMachineIn.OilPumpOk_DI && 1==gMachineInfo.OilPumpDelayDone && 0== gMachineInfo.Auto)) //ipis0222 Pump start finish
		{
			if(IPT2_ACC_Extrlift_P.y !=0)
			{
				if(1==	gMachineInfo.bAccuPump_Extrlift_Calib)
				{
					//	gUserPara.AccuPressure_Calib = gMachineFix.OilAccu.AccuPressure10V/IPT2_ACC_Extrlift_P.y;
					//gUserPara.AccuPressure_Calib = IPT2_ACC_Extrlift_P.y;
					gUserFix_new.AccuPressure_Extrlift_Calib = IPT2_ACC_Extrlift_P.y;
				}
			}
		}
	}
	else
	{
		if ((1==gMachineIn.OilPumpOk_DI && 0== gMachineInfo.Auto)) //ipis0222 Pump start finish
		{
			if(IPT2_ACC_Extrlift_P.y !=0)
			{
				if( 1 == gMachineInfo.bAccuPump_Extrlift_Calib)
				{
					//	gUserPara.AccuPressure_Extrlift_Calib = gMachineFix.OilAccu_Extrlift.AccuPressure10V/IPT2_ACC_Extrlift_P.y;
					//gUserPara.AccuPressure_Extrlift_Calib = IPT2_ACC_Extrlift_P.y;
					gUserFix_new.AccuPressure_Extrlift_Calib = IPT2_ACC_Extrlift_P.y;

				}
			}
		}
	}

	if ((0== gMachineInfo.Auto)) //ipis0222 Pump start finish
	{
		if(1 == gMachineInfo.bAccuPump_Extrlift_MinCalib)
		{
			//	gUserPara.AccuPumpMinCalib = IPT2_ACC_Extrlift_P.y;
			gUserFix_new.AccuPump_Extrlift_MinCalib = IPT2_ACC_Extrlift_P.y;
		}
	}
	if (IPT2_ACC_Extrlift_P.y-gUserFix_new.AccuPump_Extrlift_MinCalib >=0)
	{
		if (0!=(gUserFix_new.AccuPressure_Extrlift_Calib - gUserFix_new.AccuPump_Extrlift_MinCalib))  //ipis1207
		{
			gMachineInfo.OilAccuPressure_Extrlift=(IPT2_ACC_Extrlift_P.y-gUserFix_new.AccuPump_Extrlift_MinCalib)*((gMachineFix.OilAccu_Extrlift.AccuPressure10V-gUserFix_new.AccuPressure_Extrlift_0V)/(gUserFix_new.AccuPressure_Extrlift_Calib-gUserFix_new.AccuPump_Extrlift_MinCalib));
		}
	}
	else
	{
		gMachineInfo.OilAccuPressure_Extrlift =0;
	}

	/*--------------------------------------------------------------------------------------------------------------------*/

	/*---------------Servo Flow----------------*/

	OilFluxNode[0].X = gUserFix.iMinFluxV;
	OilFluxNode[1].X = gUserFix.iMaxFluxV;

	OilFluxNode[0].Y = gUserFix.rMinServoFlow;
	OilFluxNode[1].Y = gUserFix.rMaxServoFlow;

	LinSplineOilFlux.Update = gRecipeOperate.OnceSave;

	IPT2_OilFlux.u = gHardWare.AI4632_1[3];

	/* call function block */
	HydPT2(&IPT2_OilFlux);

	gMachineInfo.aiOilFlux = (int)(IPT2_OilFlux.y  * 100/32767) ;

	LinSplineOilFlux.x = IPT2_OilFlux.y;

	HCRLinSpline(&LinSplineOilFlux);

	//	gMachineInfo.aiOilFlux = LinSplineOilFlux.y;

	//	OilFluxNode[0].X =
	//
	//	OilFluxNode[0].Y =

}/* end of cyclic   */
```

#### difilter.c
```c
#ifdef _DEFAULT_INCLUDES
	#include <AsDefault.h>
#endif

/*****************************   DI filter  ***************************************/
void DIFilter(DI_Filter_typ * pDI)
{
	unsigned long	BaseTimes;
	if(0 == pDI->tTime)pDI->tTime = 200;                /*  ms  */
	if(0 == pDI->Percent)pDI->Percent = 80;           /*  0 -- 100 */
	if(pDI->TC_Time != 0 && pDI->tTime > 2 * pDI->TC_Time)
	{
		BaseTimes = pDI->tTime/pDI->TC_Time;
		pDI->TimeCounter++;
		if(pDI->TimeCounter > 100 * BaseTimes)pDI->TimeCounter = pDI->TimeCounter - 100 * BaseTimes;

		if(pDI->In != 0)
		{
			pDI->Counter++;
		}

		if(0 == (pDI->TimeCounter % BaseTimes))
		{
			if(	pDI->Counter > BaseTimes * pDI->Percent /100)
			{
				pDI->Out = 1;
			}
			else
			{
				pDI->Out = 0;
			}
			pDI->Counter = 0;
		}
	}
	else
	{
		if(pDI->In != 0)
		{
			pDI->Out = 1;
		}
		else
		{
			pDI->Out = 0;
		}
	}
}
```

#### tk1_in.var
```iecst
VAR
	tTask : REAL := 0.0;
	RTInfo_Task : RTInfo := (0);
	LCarriageFilter : HydMovAvgFlt;
	RCarriageFilter : HydMovAvgFlt;
	LClampFilter : HydMovAvgFlt;
	RClampFilter : HydMovAvgFlt;
	LBlowpinFilter : HydMovAvgFlt;
	RBlowpinFilter : HydMovAvgFlt;
	ServoFilter : HydMovAvgFlt;
	lPT2_MeltP_A : HydPT2;
	lPT2_MeltP_B : HydPT2;
END_VAR
(*Extruder A*)
VAR
	DISpeedExtrA : BOOL;
	vActHydDT2ExtrA : HydDT2;
	RotatespeedExtrA : INT;
END_VAR
(*Extruder B*)
VAR
	DISpeedExtrB : BOOL;
	vActHydDT2ExtrB : HydDT2;
	RotatespeedExtrB : INT;
END_VAR
(*Extruder C*)
VAR
	DISpeedExtrC : BOOL;
	vActHydDT2ExtrC : HydDT2;
	RotatespeedExtrC : INT;
END_VAR
(*Extruder D*)
VAR
	DISpeedExtrD : BOOL;
	vActHydDT2ExtrD : HydDT2;
	RotatespeedExtrD : INT;
END_VAR
(*Extruder Visu*)
VAR
	DISpeedExtrVisu : BOOL;
	vActHydDT2ExtrVisu : HydDT2;
	RotatespeedExtrVisu : INT;
	IPT2_ACC_P : HydPT2;
	IPT2_OilFlux : HydPT2; (*Calculate servo flow from inverter*)
	LinSplineOilFlux : HCRLinSpline;
	OilFluxNode : ARRAY[0..1] OF HCRNode_typ;
	IPT2_ACC_Extrlift_P : HydPT2;
END_VAR
```

- edge.h (reference to Logical/GlobalIncludes/edge.h)

### Program Logical/In_Out/tk1_out (ANSIC, version 1.00.0) - task 1 fast output

#### tk1_out.c
```c
/********************************************************************
 * COPYRIGHT --  B&R China
 ********************************************************************
 * Program: tk1_out
 * File: tk1_out.c
 * Author: lijianjun
 * Created: March 06, 2013
 ********************************************************************
 * Implementation of program tk1_out --- task 1 # output
 ********************************************************************/

#include <bur/plctypes.h>

#ifdef _DEFAULT_INCLUDES
#include <AsDefault.h>
#endif

#include "pic_id.h"
//#include "keyap880.h"
#include "keyap2100.h"

#define  ABS(X)           (((X) > 0.0) ? (X) : (-1.0*(X)))
/*************************************************************************************
     	        		I N I T U P  O F   T H E   T A S K
*************************************************************************************/
_INIT void init ( void )
{
	RTInfo_Task.enable = 1;
	RTInfo(&RTInfo_Task);

	tTask = RTInfo_Task.cycle_time/1000.0/1000.0;		/*  from us ---> s  */

	ExtrA_Ramp.Ts = tTask;
	ExtrB_Ramp.Ts = tTask;
	ExtrV_Ramp.Ts = tTask;
	fubP_Ramp.Ts  = tTask;

	gHardWare.AOForceNum = 19;

	gMachineOut.P_Test = 0.0;
	gMachineOut.Q_Test = 0.0;

}/* _INIT void init ( void )  */
/**************************************************************************************
****				C Y C L I C   P A R T   O F   T H E   T A S K  				   ****
**************************************************************************************/
_CYCLIC void cyclic ( void )
{

	/* --------------------- A extruder ramp function  --------------------- */
	//	if(gExtruderA.Step != 200)
	//	{
	//		ExtrA_Ramp.Accel = gMachineFix.ExtruderA.Accel;
	//	}
	//	else
	//	{
	//		ExtrA_Ramp.Accel = 1000;
	//	}
	//	if(ExtrA_Ramp.Accel == 0.0)ExtrA_Ramp.Accel = 10.0; /* 10 %/s  */
	//	ExtrA_Ramp.Set = gExtruderA.Out;
	//
	//	/* call function */
	//	HydRampCos(&ExtrA_Ramp);
	//
	//	gExtruderA.ActSpeed  = ExtrA_Ramp.Out;
	//
	//	gHardWare.AO4632_1[0] = (INT)(ExtrA_Ramp.Out * 327.67) ;

	/* --------------------- B extruder ramp function  --------------------- */
	//	if(gExtruderB.Step != 200)
	//	{
	//		ExtrB_Ramp.Accel = gMachineFix.ExtruderB.Accel;
	//	}
	//	else
	//	{
	//		ExtrB_Ramp.Accel = 1000;
	//	}
	//	if(ExtrB_Ramp.Accel == 0.0)ExtrB_Ramp.Accel = 10.0; /* 10%/s  */
	//	ExtrB_Ramp.Set = gExtruderB.Out;
	//
	//	HydRampCos(&ExtrB_Ramp);
	//
	//	gExtruderB.ActSpeed  = ExtrB_Ramp.Out;
	//
	//	gHardWare.AO4632_1[3] = (INT)(ExtrB_Ramp.Out * 327.67) ;

	//	if(3 == gHardWare.AOForceNum)gHardWare.AO4632_1[3]  = gHardWare.AOForce[3];

	/* --------------------- visual extruder ramp function  --------------------- */
	//	ExtrV_Ramp.Accel = gMachineFix.ExtruderVisu.Accel;
	//	if(ExtrV_Ramp.Accel == 0.0)ExtrV_Ramp.Accel = 100.0; /* 100 RPM/s  */
	//	ExtrV_Ramp.Set = gExtruderVisu.Out;
	//
	//	HydRampCos(&ExtrV_Ramp);
	//
	//	gExtruderVisu.ActSpeed  = ExtrV_Ramp.Out;

	/*------------------C Extruder Ao ouput for color contorl---------------*/

	//	gHardWare.AO4622_1[3] = gExtruderCCtrl.aoSetSpeed;

	/* ------------------------------------------------------------------------------ */
	/* --------------  Servo pump / System Prop valve pressure   -------------------- */
	/* ------------------------------------------------------------------------------ */
	if(1 == gMachineInfo.Auto)
	{
		gMachineOut.P_Test = 0.0;
		gMachineOut.Q_Test = 0.0;
		gMachineOut.P_Test2 = 0.0;
		gMachineOut.Q_Test2 = 0.0;
	}

	rMaxP = 0.0;
	rMaxP2 = 0.0;

	/*--------------------------------*/
	/*--------First Pressure---------*/
	/*--------------------------------*/
	if ((1==gMachineIn.OilPumpOk_DI && 1==gMachineInfo.OilPumpDelayDone && 0== gMachineInfo.Auto)) //ipis0222 Pump start finish
	{
		if((rMaxP < gMachineOut.P_Test) && (PIC_IO_AO_1 == gPanelObj.GetPicture|| PIC_PRESSURE_CALIBRATION == gPanelObj.GetPicture ) && (1 == btnTesetPQ))
		{
			rMaxP = gMachineOut.P_Test;
		}
	}
	else
	{
		btnTesetPQ = 0;
	}

	//蓄壓器補壓壓力
	if(rMaxP < gMachineOut.P_Charge)
	{
		rMaxP =	gMachineOut.P_Charge;
	}

	//抬頭蓄壓器補壓壓力
	if(rMaxP < gMachineOut.P_Charge_Extrlift)
	{
		rMaxP =	gMachineOut.P_Charge_Extrlift;
	}

	if(rMaxP < RMold.Lock.p_set)
	{
		rMaxP = RMold.Lock.p_set;
	}

	//Clamp
	if( PRESSURE_OUTPUT_SYSTEM_SINGLE == gMachineFix.MoldR.Clamp.ePressueOutputType)
	{
		if(rMaxP < RMold.Clamp.p_set)
		{
			rMaxP = RMold.Clamp.p_set;
		}
	}

	//Carriage
	if( PRESSURE_OUTPUT_SYSTEM_SINGLE == gMachineFix.MoldR.Carriage.ePressueOutputType)
	{
		if(rMaxP < RMold.Carriage.p_set)
		{
			rMaxP = RMold.Carriage.p_set;
		}
	}

	//Blowpin
	if( PRESSURE_OUTPUT_SYSTEM_SINGLE == gMachineFix.MoldR.BlowPin.ePressueOutputType)
	{
		if(rMaxP < RMold.BlowPin.p_set)
		{
			rMaxP = RMold.BlowPin.p_set;
		}
	}

	//Submold . Bottom Submold
	if( PRESSURE_OUTPUT_SYSTEM_SINGLE == gMachineFix.MoldR.SubMold.ePressueOutputType)
	{
		if(rMaxP < RMold.SubMold.p_set)
		{
			rMaxP = RMold.SubMold.p_set;
		}
		if(rMaxP < RMold.BottomSubMold.p_set)
		{
			rMaxP = RMold.BottomSubMold.p_set;
		}
	}

	//TopDeflash
	if( PRESSURE_OUTPUT_SYSTEM_SINGLE == gMachineFix.MoldR.TopDeflash.ePressueOutputType)
	{
		if(rMaxP < RMold.TopDeflash.p_set)
		{
			rMaxP = RMold.TopDeflash.p_set;
		}
	}

	//BottomDeflash
	if( PRESSURE_OUTPUT_SYSTEM_SINGLE == gMachineFix.MoldR.BottomDeflash.ePressueOutputType)
	{
		if(rMaxP < RMold.BottomDeflash.p_set)
		{
			rMaxP = RMold.BottomDeflash.p_set;
		}
	}

	//RobotTransfer
	if( PRESSURE_OUTPUT_SYSTEM_SINGLE == gMachineFix.MoldR.RobotTransfer.ePressueOutputType)
	{
		if(rMaxP < RMold.Robot.Transfer.p_set)
		{
			rMaxP = RMold.Robot.Transfer.p_set;
		}
	}

	/*--------------------------------*/
	/*--------Second Pressure---------*/
	/*--------------------------------*/
	if ((1==gMachineIn.OilPumpOk_DI && 1==gMachineInfo.OilPumpDelayDone && 0== gMachineInfo.Auto)) //ipis0222 Pump start finish
	{
		if((rMaxP2 < gMachineOut.P_Test2) && (PIC_IO_AO_1 == gPanelObj.GetPicture || PIC_PRESSURE_CALIBRATION == gPanelObj.GetPicture ) && (1 == btnTesetPQ))
		{
			rMaxP2 = gMachineOut.P_Test2;
			//		gMachineOut.LMold.MovementValve = btnTesetPQ;
		}
	}
	else
	{
		btnTesetPQ=0;
	}

	//Clamp
	if( PRESSURE_OUTPUT_SYSTEM_SINGLE == gMachineFix.MoldL.Clamp.ePressueOutputType)
	{
		if(rMaxP2 < LMold.Clamp.p_set)
		{
			rMaxP2 = LMold.Clamp.p_set;
		}
	}

	//Carriage
	if( PRESSURE_OUTPUT_SYSTEM_SINGLE == gMachineFix.MoldL.Carriage.ePressueOutputType)
	{
		if(rMaxP2 < LMold.Carriage.p_set)
		{
			rMaxP2 = LMold.Carriage.p_set;
		}
	}

	//Blowpin
	if( PRESSURE_OUTPUT_SYSTEM_SINGLE == gMachineFix.MoldL.BlowPin.ePressueOutputType)
	{
		if(rMaxP2 < LMold.BlowPin.p_set)
		{
			rMaxP2 = LMold.BlowPin.p_set;
		}
	}

	//Submold . Bottom Submold
	if( PRESSURE_OUTPUT_SYSTEM_SINGLE == gMachineFix.MoldL.Carriage.ePressueOutputType)
	{
		if(rMaxP2 < LMold.SubMold.p_set)
		{
			rMaxP2 = LMold.SubMold.p_set;
		}
		if(rMaxP2 < LMold.BottomSubMold.p_set)
		{
			rMaxP2 = LMold.BottomSubMold.p_set;
		}
	}

	//TopDeflash
	if( PRESSURE_OUTPUT_SYSTEM_SINGLE == gMachineFix.MoldL.TopDeflash.ePressueOutputType)
	{
		if(rMaxP2 < LMold.TopDeflash.p_set)
		{
			rMaxP2 = LMold.TopDeflash.p_set;
		}
	}

	//BottomDeflash
	if( PRESSURE_OUTPUT_SYSTEM_SINGLE == gMachineFix.MoldL.BottomDeflash.ePressueOutputType)
	{
		if(rMaxP2 < LMold.BottomDeflash.p_set)
		{
			rMaxP2 = LMold.BottomDeflash.p_set;
		}
	}

	//RobotTransfer
	if( PRESSURE_OUTPUT_SYSTEM_SINGLE == gMachineFix.MoldL.RobotTransfer.ePressueOutputType)
	{
		if(rMaxP2 < LMold.Robot.Transfer.p_set)
		{
			rMaxP2 = LMold.Robot.Transfer.p_set;
		}
	}

	/*-------------------Special-------------------------------*/

	if( PRESSURE_OUTPUT_SYSTEM_SINGLE == gMachineFix.Plate.ePressueOutputType )
	{
		/*-------Plate Up Down AO L------*/
		if ( 5000== RMold.Plate.Step  || 15000==RMold.Plate.Step || 5000== LMold.Plate.Step  || 15000==LMold.Plate.Step )
		{
			if(1 == gMachineFix.Plate.bUpDnPressureOutputLeft)
			{
				if(rMaxP2 < LMold.Plate.p_set)
				{
					rMaxP2 = LMold.Plate.p_set;
				}
				if(rMaxP2 < RMold.Plate.p_set)
				{
					rMaxP2 = RMold.Plate.p_set;
				}

			}
			else
			{
				if(rMaxP < LMold.Plate.p_set)
				{
					rMaxP = LMold.Plate.p_set;
				}
				if(rMaxP < RMold.Plate.p_set)
				{
					rMaxP = RMold.Plate.p_set;
				}

			}
		}

		/*-------Plate Fw Bw AO R------*/
		if (6200 == RMold.Plate.Step ||16200 == RMold.Plate.Step  ||6200 == LMold.Plate.Step ||16200 == LMold.Plate.Step
			||(RMold.Plate.Step >=6500&& RMold.Plate.Step <=6520 ) ||(LMold.Plate.Step >=6500&& LMold.Plate.Step <=6520)) //ipis0305
		{
			if(1 == gMachineFix.Plate.bFwBwPressureOutputLeft)
			{
				if(rMaxP2 < LMold.Plate.p_set)
				{
					rMaxP2 = LMold.Plate.p_set;
				}
				if(rMaxP2 < RMold.Plate.p_set)
				{
					rMaxP2 = RMold.Plate.p_set;
				}
			}
			else
			{
				if(rMaxP < LMold.Plate.p_set)
				{
					rMaxP = LMold.Plate.p_set;
				}
				if(rMaxP < RMold.Plate.p_set)
				{
					rMaxP = RMold.Plate.p_set;
				}
			}
		}
	}

	/*--------------------------------------------------------*/

	/* clean valve  */
	if(1 == gMacTimer.ValveCleanTotal.IN || 1 == gMachineInfo.Calib)
	{
		if(1 == gMachineOut.ValveFw || 1 == gMachineOut.ValveBw)
		{
			if(rMaxP < gMachineFix.Pump.P_CleanValve)rMaxP = gMachineFix.Pump.P_CleanValve;
		}
	}

	/* Auto running */
	if(1 == gMachineInfo.Auto)
	{
		//		if(rMaxP < gMachineFix.Pump.P_Idle)rMaxP = gMachineFix.Pump.P_Idle;
	}

	if(RMold.Carriage.v_set != 0 || LMold.Carriage.v_set != 0)
	{
		//		if(rMaxP < 1.0)rMaxP = gMachineFix.Pump.P_Idle;
	}

	/*---------------Pump Pressure------------------*/
	/* Auto running */
	if(rMaxP > gMachineFix.Pump.MaxP1)rMaxP = gMachineFix.Pump.MaxP1;
	if(rMaxP2 > gMachineFix.Pump.MaxP2) rMaxP2 = gMachineFix.Pump.MaxP2;
	/* Default value */
	if(gMachineFix.Pump.accel_P < 100)gMachineFix.Pump.accel_P = 1000;

	/*--First Pressure (Right)--*/
	fubP_Ramp.Set = rMaxP;
	fubP_Ramp.Accel = gMachineFix.Pump.accel_P;
	HydRampCos(&fubP_Ramp);
	aoPressure = fubP_Ramp.Out * 32767/gMachineFix.Pump.MaxP1;

	gMachineOut.P_Set = aoPressure / 327.67;
	gMachineOut.P_Act = aoPressure / 3276.7;
	gHardWare.AO4632_1[0] = aoPressure;

	/*--Second Pressure (Left)--*/
	fubP2_Ramp.Set = rMaxP2;
	fubP2_Ramp.Accel = gMachineFix.Pump.accel_P;
	/* Call function */
	HydRampCos(&fubP2_Ramp);

	aoPressure2 = fubP2_Ramp.Out * 32767/gMachineFix.Pump.MaxP2;

	gMachineOut.P_Set2 = aoPressure2 / 327.67;
	gMachineOut.P_Act2 = aoPressure2 / 3276.7;
	//	gHardWare.AO4632_1[1] = aoPressure2;

	/* ------------------------------------------------------------------------------ */
	/* ----------------------------    Servo pump flux     -------------------------- */
	/* ------------------------------------------------------------------------------ */

	/*---------------Servo pump flux------------------*/

	rMaxQ = 0.0;
	rMaxQ2 = 0.0;

	/*--------------------------------*/
	/*--------First Flux--------------*/
	/*--------------------------------*/
	if ((1==gMachineIn.OilPumpOk_DI && 1==gMachineInfo.OilPumpDelayDone && 0== gMachineInfo.Auto)) //ipis0222 Pump start finish
	{
		if((rMaxQ < gMachineOut.Q_Test * 327.67) && (PIC_IO_AO_1 == gPanelObj.GetPicture|| PIC_PRESSURE_CALIBRATION == gPanelObj.GetPicture ) && (1 == btnTesetPQ))
		{
			rMaxQ = gMachineOut.Q_Test * 327.67;
		}
	}

	//蓄壓器補壓流量
	if(rMaxQ < gMachineOut.Q_Charge * 327.67)
	{
		rMaxQ = gMachineOut.Q_Charge * 327.67;
	}

	//抬頭蓄壓器補壓流量
	/*output for charge Extrlift acc pump*/
	if(rMaxQ < gMachineOut.Q_Charge_Extrlift * 327.67)
	{
		rMaxQ = gMachineOut.Q_Charge_Extrlift * 327.67;
	}

	//	if(rMaxQ < ABS(RMold.Lock.aoPropValve))
	//	{
	//		rMaxQ = ABS(RMold.Lock.aoPropValve);
	//	}

	//	if(rMaxQ < ABS(LMold.Lock.aoPropValve))
	//	{
	//		rMaxQ = ABS(LMold.Lock.aoPropValve);
	//	}

	//Clamp
	if(FLUX_OUTPUT_SYSTEM_SINGLE == gMachineFix.MoldR.Clamp.eFluxOutputType)
	{
		if (rMaxQ < ABS(RMold.Clamp.v_set * 32.767))	/* ProfGen.v_set 0-1000*/
		{
			rMaxQ = ABS(RMold.Clamp.v_set * 32.767);
		}
	}

	//Carriage
	if(FLUX_OUTPUT_SYSTEM_SINGLE == gMachineFix.MoldR.Carriage.eFluxOutputType)
	{
		if (rMaxQ < ABS(RMold.Carriage.v_set * 32.767))	/* ProfGen.v_set 0-1000*/
		{
			rMaxQ = ABS(RMold.Carriage.v_set * 32.767);
		}
	}

	//BlowPin
	if(FLUX_OUTPUT_SYSTEM_SINGLE == gMachineFix.MoldR.BlowPin.eFluxOutputType)
	{
		if (rMaxQ < ABS(RMold.BlowPin.v_set * 32.767))	/* ProfGen.v_set 0-1000*/
		{
			rMaxQ = ABS(RMold.BlowPin.v_set * 32.767);
		}
	}

	//TopDeflash
	if(FLUX_OUTPUT_SYSTEM_SINGLE == gMachineFix.MoldR.TopDeflash.eFluxOutputType)
	{
		if (rMaxQ < ABS(RMold.TopDeflash.v_set * 327.67))
		{
			rMaxQ = ABS(RMold.TopDeflash.v_set * 327.67);
		}
	}

	//BottomDeflash
	if(FLUX_OUTPUT_SYSTEM_SINGLE == gMachineFix.MoldR.BottomDeflash.eFluxOutputType)
	{
		if (rMaxQ < ABS(RMold.BottomDeflash.v_set * 327.67))
		{
			rMaxQ = ABS(RMold.BottomDeflash.v_set * 327.67);
		}
	}

	//RobotTransfer
	if(FLUX_OUTPUT_SYSTEM_SINGLE == gMachineFix.MoldR.RobotTransfer.eFluxOutputType)
	{
		if (rMaxQ < ABS(RMold.Robot.Transfer.v_set * 327.67))
		{
			rMaxQ = ABS(RMold.Robot.Transfer.v_set * 327.67);
		}
	}

	//Plate
	if(FLUX_OUTPUT_SYSTEM_SINGLE == gMachineFix.Plate.eFluxOutputType)
	{
		if (rMaxQ < ABS(RMold.Plate.v_set * 327.67))
		{
			rMaxQ = ABS(RMold.Plate.v_set * 327.67);
		}
	}

	/*--------------------------------*/
	/*--------Second Flux--------------*/
	/*--------------------------------*/
	if ((1==gMachineIn.OilPumpOk_DI && 1==gMachineInfo.OilPumpDelayDone && 0== gMachineInfo.Auto)) //ipis0222 Pump start finish
	{
		if((rMaxQ2 < gMachineOut.Q_Test2 * 327.67) && (PIC_IO_AO_1 == gPanelObj.GetPicture|| PIC_PRESSURE_CALIBRATION == gPanelObj.GetPicture ) && (1 == btnTesetPQ))
		{
			rMaxQ2 = gMachineOut.Q_Test2 * 327.67;
		}
	}

	//	if(rMaxQ2 < ABS(RMold.Lock.aoPropValve))
	//	{
	//		rMaxQ2 = ABS(RMold.Lock.aoPropValve);
	//	}

	//	if(rMaxQ2 < ABS(LMold.Lock.aoPropValve))
	//	{
	//		rMaxQ2 = ABS(LMold.Lock.aoPropValve);
	//	}

	//Clamp
	if(FLUX_OUTPUT_SYSTEM_SINGLE == gMachineFix.MoldR.Clamp.eFluxOutputType)
	{
		if (rMaxQ2 < ABS(LMold.Clamp.v_set * 32.767))	/* ProfGen.v_set 0-1000*/
		{
			rMaxQ2 = ABS(LMold.Clamp.v_set * 32.767);
		}
	}

	//Carriage
	if(FLUX_OUTPUT_SYSTEM_SINGLE == gMachineFix.MoldR.Carriage.eFluxOutputType)
	{
		if (rMaxQ2 < ABS(LMold.Carriage.v_set * 32.767))	/* ProfGen.v_set 0-1000*/
		{
			rMaxQ2 = ABS(LMold.Carriage.v_set * 32.767);
		}
	}

	//BlowPin
	if(FLUX_OUTPUT_SYSTEM_SINGLE == gMachineFix.MoldR.BlowPin.eFluxOutputType)
	{
		if (rMaxQ2 < ABS(LMold.BlowPin.v_set * 32.767))	/* ProfGen.v_set 0-1000*/
		{
			rMaxQ2 = ABS(LMold.BlowPin.v_set * 32.767);
		}
	}

	//TopDeflash
	if(FLUX_OUTPUT_SYSTEM_SINGLE == gMachineFix.MoldR.TopDeflash.eFluxOutputType)
	{
		if (rMaxQ2 < ABS(LMold.TopDeflash.v_set * 327.67))
		{
			rMaxQ2 = ABS(LMold.TopDeflash.v_set * 327.67);
		}
	}

	//BottomDeflash
	if(FLUX_OUTPUT_SYSTEM_SINGLE == gMachineFix.MoldR.BottomDeflash.eFluxOutputType)
	{
		if (rMaxQ2 < ABS(LMold.BottomDeflash.v_set * 327.67))
		{
			rMaxQ2 = ABS(LMold.BottomDeflash.v_set * 327.67);
		}
	}

	//RobotTransfer
	if(FLUX_OUTPUT_SYSTEM_SINGLE == gMachineFix.MoldR.RobotTransfer.eFluxOutputType)
	{
		if (rMaxQ2 < ABS(LMold.Robot.Transfer.v_set * 327.67))
		{
			rMaxQ2 = ABS(LMold.Robot.Transfer.v_set * 327.67);
		}
	}

//	//Plate
//	if(FLUX_OUTPUT_SYSTEM_SINGLE == gMachineFix.Plate.eFluxOutputType)
//	{
//		if (rMaxQ2 < ABS(LMold.Plate.v_set * 327.67))
//		{
//			rMaxQ2 = ABS(LMold.Plate.v_set * 327.67);
//		}
//	}

	/*----------------------------------------------*/
	/*---------------Pump Flux Out------------------*/
	/*----------------------------------------------*/

	/*-----First Flux------*/
	if(rMaxQ > 32767)rMaxQ = 32767;
	aoFlux = (INT)rMaxQ;
	gMachineOut.Q_Set = aoFlux / 327.67;

	gHardWare.AO4632_1[1] = (INT)aoFlux;
//	gHardWare.AO4622_1[1] = aoFlux;

	/*-----Second Flux------*/
	if(rMaxQ2 > 32767)rMaxQ2 = 32767;
	aoFlux2 = (INT)rMaxQ2;
	gMachineOut.Q_Set2 = aoFlux2 / 327.67;

	//	gHardWare.AO4632_1[3] = (INT)aoFlux2;
	//	gHardWare.AO4622_1[1] = aoFlux2;

	/* ------------------------------------------------------------------------------ */
	/* ---------------------------- thickness valve output -------------------------- */
	/* ------------------------------------------------------------------------------ */

		if(1 == gMachineOut.ParisonPump)
		{
			gHardWare.AO4632_1[2] = -gThickIO.ServoOut;/*Test*/
		}
		else
		{
			gHardWare.AO4632_1[2]  = 0;
		}

	/* ------------------------------------------------------------------------------ */
	/*  ----------------------------- Flux Prop Valve  ------------------------------ */
	/* ------------------------------------------------------------------------------ */

	/* ----------------------*/
	/* ---------right--------*/
	/* ----------------------*/
	//Clamp
	if( FLUX_OUTPUT_PROP_VALVE_SINGLE == gMachineFix.MoldR.Clamp.eFluxOutputType)
	{
		//		gHardWare.AO4632_3[0] = RMold.Clamp.aoPropValve;
	}

	//Carriage
	if( FLUX_OUTPUT_PROP_VALVE_SINGLE == gMachineFix.MoldR.Carriage.eFluxOutputType)
	{
		//		gHardWare.AO4622_3[2] = RMold.Carriage.aoPropValve;
	}

	//BlowPin
	if( FLUX_OUTPUT_PROP_VALVE_SINGLE == gMachineFix.MoldR.BlowPin.eFluxOutputType)
	{
		//		gHardWare.AO4622_3[2] = RMold.BlowPin.aoPropValve;
	}

	/* ----------------------*/
	/* ---------right--------*/
	/* ----------------------*/

	//Clamp
	if( FLUX_OUTPUT_PROP_VALVE_SINGLE == gMachineFix.MoldL.Clamp.eFluxOutputType)
	{
		//		gHardWare.AO4632_3[1] = RMold.Clamp.aoPropValve;
	}

	//Carriage
	if( FLUX_OUTPUT_PROP_VALVE_SINGLE == gMachineFix.MoldL.Carriage.eFluxOutputType)
	{
		//		gHardWare.AO4622_3[2] = RMold.Carriage.aoPropValve;
	}

	//BlowPin
	if( FLUX_OUTPUT_PROP_VALVE_SINGLE == gMachineFix.MoldL.BlowPin.eFluxOutputType)
	{
		//		gHardWare.AO4622_3[2] = RMold.BlowPin.aoPropValve;
	}

	/* ------------------------------------------------------------------------------ */
	/* -------------------------- right temp SCR die lip---------------------------- */
	/* ------------------------------------------------------------------------------ */
	if(0 == gMachineOut.HeatPower)
	{
		bEnableRightDie = 0;
	}
	else if(oldHeatPower != gMachineOut.HeatPower)
	{
		bEnableRightDie = gMachineOut.HeatPower;
	}

	if(bEnableRightDie)
	{

		if(gMachineInfo.bLoweringFlag) gMachineOut.aoRightDieLipTemp = (INT)(gUserPara.RightDieLipTempSCR - gUserPara.DieLipTempSCR_Lower);
		else gMachineOut.aoRightDieLipTemp = (INT)gUserPara.RightDieLipTempSCR;
	}
	else
	{
		gMachineOut.aoRightDieLipTemp = 0;
	}

	if(gMachineOut.aoRightDieLipTemp <= 0) gMachineOut.aoRightDieLipTemp = 0;
	gHardWare.AO4632_2[0] = gMachineOut.aoRightDieLipTemp;

	/* ------------------------------------------------------------------------------ */
	/* -------------------------- left temp SCR die lip---------------------------- */
	/* ------------------------------------------------------------------------------ */
	if(0 == gMachineOut.HeatPower)
	{
		bEnableLeftDie = 0;
	}
	else if(oldHeatPower != gMachineOut.HeatPower)
	{
		bEnableLeftDie = gMachineOut.HeatPower;
	}

	if(bEnableLeftDie)
	{

		if(gMachineInfo.bLoweringFlag) gMachineOut.aoLiftDieLipTemp = (INT)(gUserPara.LiftDieLipTempSCR - gUserPara.DieLipTempSCR_Lower);
		else gMachineOut.aoLiftDieLipTemp = (INT)gUserPara.LiftDieLipTempSCR;
	}
	else
	{
		gMachineOut.aoLiftDieLipTemp = 0;
	}

	if(gMachineOut.aoLiftDieLipTemp <= 0) gMachineOut.aoLiftDieLipTemp = 0;
	gHardWare.AO4632_2[1] = gMachineOut.aoLiftDieLipTemp;

	/* ------------------------------------------------------------------------------ */
	/* --------------------------  temp SCR die lip_3    ---------------------------- */
	/* ------------------------------------------------------------------------------ */
	if(0 == gMachineOut.HeatPower)
	{
		bEnableDie3 = 0;
	}
	else if(oldHeatPower != gMachineOut.HeatPower)
	{
		bEnableDie3 = gMachineOut.HeatPower;
	}

	if(bEnableDie3)
	{
		if(gMachineInfo.bLoweringFlag) gMachineOut.aoDieLipTemp3 = (INT)(gUserPara.DieLipTempSCR3 - gUserPara.DieLipTempSCR_Lower);
		else gMachineOut.aoDieLipTemp3 = (INT)gUserPara.DieLipTempSCR3;
	}
	else
	{
		gMachineOut.aoDieLipTemp3 = 0;
	}

	if(gMachineOut.aoDieLipTemp3 <= 0) gMachineOut.aoDieLipTemp3 = 0;
	gHardWare.AO4632_2[2] = gMachineOut.aoDieLipTemp3;

	/* ------------------------------------------------------------------------------ */
	/* -------------------------- temp SCR die lip_4     ---------------------------- */
	/* ------------------------------------------------------------------------------ */
	if(0 == gMachineOut.HeatPower)
	{
		bEnableDie4 = 0;
	}
	else if(oldHeatPower != gMachineOut.HeatPower)
	{
		bEnableDie4 = gMachineOut.HeatPower;
	}

	if(bEnableDie4)
	{
		if(gMachineInfo.bLoweringFlag) gMachineOut.aoDieLipTemp4 = (INT)(gUserPara.DieLipTempSCR4 - gUserPara.DieLipTempSCR_Lower);
		else gMachineOut.aoDieLipTemp4 = (INT)gUserPara.DieLipTempSCR4;
	}
	else
	{
		gMachineOut.aoDieLipTemp4 = 0;
	}

	if(gMachineOut.aoDieLipTemp4 <= 0) gMachineOut.aoDieLipTemp4 = 0;
	gHardWare.AO4632_2[3] = gMachineOut.aoDieLipTemp4;

	/* ------------------------------------------------------------------------------ */
	/* ------------------------- temp SCR die lip Common ---------------------------- */
	/* ------------------------------------------------------------------------------ */
	if( (gMachineFix.Option.bDieLip[0] &&(0 == gUserPara.RightDieLipTempSCR || 0 == bEnableRightDie))||
		(gMachineFix.Option.bDieLip[1] &&(0 == gUserPara.LiftDieLipTempSCR || 0 == bEnableLeftDie))	||
		(gMachineFix.Option.bDieLip[2] &&(0 == gUserPara.DieLipTempSCR3 || 0 == bEnableDie3))||
		(gMachineFix.Option.bDieLip[3] &&(0 == gUserPara.DieLipTempSCR4 || 0 == bEnableDie4)))
	{
		gMachineInfo.DieLipTempLow = 1;
	}
	else
	{
		gMachineInfo.DieLipTempLow = 0;
	}

	/* ------------------------------------------------------------------------------ */
	/* -------------------- hot cutter heating  熱切刀    --------------------------- */
	/* ------------------------------------------------------------------------------ */

	if(1 == gMachineFix.Option.bCutterHeating &&  1 == gMacOption.Cutter && 1 == gMachineOut.ExtrA_On)
	{
		if(bEnableCutterHeating)
		{
			gMachineOut.CutterHeating = (INT)gUserPara.CutterHeatingSCR;
		}
		else
		{
			gMachineOut.CutterHeating = 0;
		}
	}
	else
	{
		if( 1 == bEnableCutterHeating)
		{
			gImply.NoFunction = !gMacOption.Cutter;
			gImply.FrequencyNotOn = !gMachineOut.ExtrA_On;

		}

		bEnableCutterHeating = 0;
		gMachineOut.CutterHeating = 0;
	}
	if(gMachineOut.CutterHeating <= 0) gMachineOut.CutterHeating = 0;
	gHardWare.AO4632_1[3] = gMachineOut.CutterHeating;

	oldHeatPower = gMachineOut.HeatPower;
	/* ------------------------------------------------------------------------------ */
	/*  ----------------------------- Extruder AO ----------------------------------- */
	/* ------------------------------------------------------------------------------ */

	if(CTRL_VF == gMachineFix.ExtruderA.eCtrlType )// Analog VF Control
	{
		// Extruder A
		gHardWare.AO4632_3[3] = gExtruderA.aoSetRPM;
		// Extruder B
		gHardWare.AO4632_4[2] = gExtruderB.aoSetRPM;
		// Extruder C
		gHardWare.AO4632_4[3] = gExtruderC.aoSetRPM;
		// Extruder D
		gHardWare.AO4632_4[0] = gExtruderD.aoSetRPM;
		// Extruder Visu
		gHardWare.AO4632_4[1] = gExtruderVisu.aoSetRPM;
	}

	/* --------------------------------  AO Force-------------------------------- */
	//	if(1 == gHardWare.AOForceNum[0])gHardWare.AO4632_1[0]  = gHardWare.AOForce[0];
	//	if(1 == gHardWare.AOForceNum[1])gHardWare.AO4632_1[1]  = gHardWare.AOForce[1];
	//	if(1 == gHardWare.AOForceNum[2])gHardWare.AO4632_1[2]  = gHardWare.AOForce[2];
	//	if(1 == gHardWare.AOForceNum[3])gHardWare.AO4632_1[3]  = gHardWare.AOForce[3];
	//	if(1 == gHardWare.AOForceNum[4])gHardWare.AO4632_2[0]  = gHardWare.AOForce[4];
	//	if(1 == gHardWare.AOForceNum[5])gHardWare.AO4632_2[1]  = gHardWare.AOForce[5];
	//	if(1 == gHardWare.AOForceNum[6])gHardWare.AO4632_2[2]  = gHardWare.AOForce[6];
	//	if(1 == gHardWare.AOForceNum[7])gHardWare.AO4632_2[3]  = gHardWare.AOForce[7];
	//	if(1 == gHardWare.AOForceNum[8])gHardWare.AO4632_3[0]  = gHardWare.AOForce[8];
	//	if(1 == gHardWare.AOForceNum[9])gHardWare.AO4632_3[1]  = gHardWare.AOForce[9];
	//	if(1 == gHardWare.AOForceNum[10])gHardWare.AO4632_3[2]  = gHardWare.AOForce[10];/*LMold.Clamp.aoPropValve*/
	//	if(1 == gHardWare.AOForceNum[11])gHardWare.AO4632_3[3]  = gHardWare.AOForce[11];/*RMold.Clamp.aoPropValve*/

	if(0 == gHardWare.AOForceNum)gHardWare.AO4632_1[0]  = gHardWare.AOForce[0];
	if(1 == gHardWare.AOForceNum)gHardWare.AO4632_1[1]  = gHardWare.AOForce[1];
	if(2 == gHardWare.AOForceNum)gHardWare.AO4632_1[2]  = gHardWare.AOForce[2];
	if(3 == gHardWare.AOForceNum)gHardWare.AO4632_1[3]  = gHardWare.AOForce[3];

	if(4 == gHardWare.AOForceNum)gHardWare.AO4632_2[0]  = gHardWare.AOForce[4];
	if(5 == gHardWare.AOForceNum)gHardWare.AO4632_2[1]  = gHardWare.AOForce[5];
	if(6 == gHardWare.AOForceNum)gHardWare.AO4632_2[2]  = gHardWare.AOForce[6];
	if(7 == gHardWare.AOForceNum)gHardWare.AO4632_2[3]  = gHardWare.AOForce[7];

	if(8 == gHardWare.AOForceNum)gHardWare.AO4632_3[0]  = gHardWare.AOForce[8];
	if(9 == gHardWare.AOForceNum)gHardWare.AO4632_3[1]  = gHardWare.AOForce[9];
	if(10 == gHardWare.AOForceNum)gHardWare.AO4632_3[2]  = gHardWare.AOForce[10];
	if(11 == gHardWare.AOForceNum)gHardWare.AO4632_3[3]  = gHardWare.AOForce[11];

	if(12 == gHardWare.AOForceNum)gHardWare.AO4632_4[0]  = gHardWare.AOForce[12];
	if(13 == gHardWare.AOForceNum)gHardWare.AO4632_4[1]  = gHardWare.AOForce[13];
	if(14 == gHardWare.AOForceNum)gHardWare.AO4632_4[2]  = gHardWare.AOForce[14];
	if(15 == gHardWare.AOForceNum)gHardWare.AO4632_4[3]  = gHardWare.AOForce[15];

	/* ------------------------------------------------------------------------------------- */
	/* --------------------------------     Module error    -------------------------------- */
	/* ------------------------------------------------------------------------------------- */
	if(1 == gPROCESS_info.moduleErr)
	{
		gHardWare.AO4632_1[0]  = 0;
		gHardWare.AO4632_1[1]  = 0;
		gHardWare.AO4632_1[2]  = 0;
		gHardWare.AO4632_1[3]  = 0;

		gHardWare.AO4632_2[0]  = 0;
		gHardWare.AO4632_2[1]  = 0;
		gHardWare.AO4632_2[2]  = 0;
		gHardWare.AO4632_2[3]  = 0;

		gHardWare.AO4632_3[0]  = 0;
		gHardWare.AO4632_3[1]  = 0;
		gHardWare.AO4632_3[2]  = 0;
		gHardWare.AO4632_3[3]  = 0;

		gHardWare.AO4632_4[0]  = 0;
		gHardWare.AO4632_4[1]  = 0;
		gHardWare.AO4632_4[2]  = 0;
		gHardWare.AO4632_4[3]  = 0;
	}/* if(1 == gPROCESS_info.moduleErr) */
}/* end of cyclic   */
```

#### tk1_out.var
```iecst
VAR
	tTask : REAL := 0.0;
	RTInfo_Task : RTInfo := (0);
	ExtrA_Ramp : HydRampCos;
	ExtrB_Ramp : HydRampCos;
	ExtrV_Ramp : HydRampCos;
	fubP_Ramp : HydRampCos;
	fubP2_Ramp : HydRampCos;
	rMaxP : REAL;
	rMaxP2 : REAL;
	rMaxQ : REAL;
	rMaxQ2 : REAL;
	aoPressure : DINT;
	aoPressure2 : DINT;
	aoFlux : DINT;
	aoFlux2 : DINT;
	bEnableLeftDie : BOOL;
	bEnableRightDie : BOOL;
	bEnableDie3 : BOOL;
	bEnableDie4 : BOOL;
	bEnableCutterHeating : BOOL;
END_VAR
(*Extruder Speed*)
VAR
	oldHeatPower : USINT;
END_VAR
```

### Program Logical/In_Out/tk2_io (ANSIC, version 1.00.0) - mormal input and output
